FUNCTION_BLOCK FB_LamparaConmutada_SFC
// La lampara se enciende tras un determinado numero de pulsaciones
// La lampara se apaga tras accionar el pulsador de reinicio
VAR
    Pulsacion: R_TRIG;
    Lampara AT %Q*: BOOL;
    Pulsador AT %I*: BOOL;
END_VAR

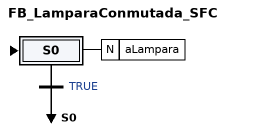
INITIAL_STEP S0:
    aLampara(N);
END_STEP
TRANSITION FROM S0 TO S0
    := TRUE;
END_TRANSITION

ACTION aLampara:
Pulsacion(CLK := Pulsador);

IF Pulsacion.Q THEN
    Lampara := NOT Lampara;
END_IF
END_ACTION

END_FUNCTION_BLOCK

(* stored: Version 1.1.0.1, ProductVersion 3.1.4024.15
   POU FB_LamparaConmutada_SFC: Id {627d8519-ef3d-4358-89ad-fa30f84c70ba}, SpecialFunc None
   Action aLampara: Id {692c89e8-9cde-44df-ba38-bfdc617d6826} *)
